(* CODESYS project mpm_jsonparser.library
   Author: Cory Tollefsrud
   Placeholder: MPM_JsonParser
   Title: MPM_JsonParser
   Version: 0.2.3.1
   Company: MatixPM

Project tree, tasks and I/O mapping:
  libraries: Base Interfaces, * (System); Tc2_System, * (Beckhoff Automation GmbH); Tc3_JsonXml, * (Beckhoff Automation GmbH)
  FUN/
    function F_Map_ST_AnyType_User [ST]
  Legecy/
    function block FB_JsonSchemaEx_OLD [ST]: M_CreateSchemaJson, M_PraseSchemaJson, M_PraseJsonSchema, M_SetJsonSchema, M_SetMemberValue, M_SetMemberValue_AnyType, M_SetMemberValueEx, M_SetMemberValueEx_AnyType, M_GetJsonMemberValue, M_GetJsonMemberValue_AnyType, M_SetJsonMember, M_SetJsonMemberValue, M_SetJsonMemberValue_AnyType, M_SetJsonMemberValueEx, M_SetJsonMemberValueEx_AnyType, M_SetJsonMemberValueNonDefault, M_SetJsonSchemaValue
  data type DUT_JsonMemberValue
  data type DUT_JsonSchema
  data type DUT_Pointers
  data type E_TypeClassEx
  function block FB_JsonEx [ST]: M_SetMemberValue, M_SetMemberValueEx, M_GetJsonMemberValue, M_SetJsonMember, M_SetJsonMemberValue, M_SetJsonMemberValueEx, M_SetJsonMemberValueNonDefault
  function block FB_JsonSchemaEx [ST]: M_CreateSchemaJson, M_PraseSchemaJson, M_RegisterSchemaObject
  function block FB_JsonSchemaExBase [ST]: M_AssignSchemaMember, M_AssignSchemaMemberEx, M_GetJsonSchemaValue, M_PraseJsonSchema, M_Read, M_SetJsonSchema, M_SetJsonSchemaValue, M_SetMemberSchemaValue, M_Write
  function block FB_JsonSchemaObject [ST]: M_AssignSchemaMember, M_AssignSchemaMemberEx, M_CreateSchemaJson, M_GetWriteStatus, M_PraseSchemaJson, M_Read, M_SetJsonRef, M_SetJsonSchemaValue, M_TriggerWrite, M_Write, P_sJsonRoot
  data type ST_AnyType_User
  data type ST_SchemaMember
*)

// DUT_JsonMemberValue
TYPE DUT_JsonMemberValue :
STRUCT
	member				: STRING(255);
	value				: STRING(10000);
END_STRUCT
END_TYPE

// DUT_JsonSchema
TYPE DUT_JsonSchema :
STRUCT
	jsonValueRoot			: REFERENCE TO sJsonValue;
	jsonValue				: sJsonValue;
	member					: STRING(255);
	typeClass				: E_TypeClassEx;
END_STRUCT
END_TYPE

// DUT_Pointers
//{attribute 'no_copy'} // used so that on that on a online change the pointers will update there address.

//This is only to copy values in and out of DOM memory
TYPE DUT_Pointers :
STRUCT
	_byteArray			: ARRAY [0..7] OF BYTE;
	pString				: POINTER TO STRING(1000); //String
	pJson				: POINTER TO STRING(10000);	//Big string
	pSint				: POINTER TO SINT;
	pInt				: POINTER TO INT;
	pUInt				: POINTER TO UINT;
	pDint				: POINTER TO DINT;
	pUDint				: POINTER TO UDINT;	
	pLint				: POINTER TO LINT;
	pUlint				: POINTER TO ULINT;	
	pBOOL				: POINTER TO BOOL;
	pLREAL				: POINTER TO LREAL;
	pREAL				: POINTER TO REAL;
	pFileTime			: POINTER TO FILETIME;
END_STRUCT
END_TYPE

// E_TypeClassEx
{attribute 'qualified_only'}

TYPE E_TypeClassEx :
(
	Type_ANY := TypeClass.TYPE_ANY,
	TYPE_ANYBIT := TypeClass.TYPE_ANYBIT,
	TYPE_ANYDATE := TypeClass.TYPE_ANYDATE,
	TYPE_ANYINT := TypeClass.TYPE_ANYINT,	
	TYPE_ANYNUM := TypeClass.TYPE_ANYNUM,	
	TYPE_ANYREAL := TypeClass.TYPE_ANYREAL,		
	TYPE_ARRAY := TypeClass.TYPE_ARRAY,	
	TYPE_BIT := TypeClass.TYPE_BIT,		
	TYPE_BITCONST := TypeClass.TYPE_BITCONST,		
	TYPE_BOOL := TypeClass.TYPE_BOOL,
	TYPE_BYTE := TypeClass.TYPE_BYTE,	
	TYPE_DATE := TypeClass.TYPE_DATE,
	TYPE_DATEANDTIME := TypeClass.TYPE_DATEANDTIME,			
	TYPE_DINT := TypeClass.TYPE_DINT,		
	TYPE_DWORD := TypeClass.TYPE_DWORD,		
	TYPE_ENUM := TypeClass.TYPE_ENUM,	
	TYPE_INT := TypeClass.TYPE_INT,	
	TYPE_INTERFACE := TypeClass.TYPE_INTERFACE,	
	TYPE_LAZY := TypeClass.TYPE_LAZY,		
	TYPE_LINT := TypeClass.TYPE_LINT,
	TYPE_LREAL := TypeClass.TYPE_LREAL,	
	TYPE_LTIME := TypeClass.TYPE_LTIME,	
	TYPE_LWORD := TypeClass.TYPE_LWORD,
	TYPE_NONE := TypeClass.TYPE_NONE,
	TYPE_PARAMS := TypeClass.TYPE_PARAMS,	
	TYPE_POINTER := TypeClass.TYPE_POINTER,	
	TYPE_REAL := TypeClass.TYPE_REAL, 	
	TYPE_REFERENCE := TypeClass.TYPE_REFERENCE,	
	TYPE_SINT := TypeClass.TYPE_SINT,	
	TYPE_STRING := TypeClass.TYPE_STRING,	
	TYPE_SUBRANGE := TypeClass.TYPE_SUBRANGE,
	TYPE_TIME := TypeClass.TYPE_TIME,			
	TYPE_TIMEOFDAY := TypeClass.TYPE_TIMEOFDAY,					
	TYPE_UDINT := TypeClass.TYPE_UDINT,		
	TYPE_UINT := TypeClass.TYPE_UINT,	
	TYPE_ULINT := TypeClass.TYPE_ULINT,
	TYPE_USERDEF := TypeClass.TYPE_USERDEF,	
	TYPE_USINT := TypeClass.TYPE_USINT,	
	TYPE_WORD := TypeClass.TYPE_WORD,	
	TYPE_WSTRING := TypeClass.TYPE_WSTRING,
	TYPE_JSON := 10000,
	TYPE_JSONARRAY := 10002,	
	TYPE_FILETIME := 10001	
)INT;
END_TYPE

// ST_AnyType_User
{attribute 'enable_dynamic_creation'}
TYPE ST_AnyType_User :
STRUCT
	//name
	name : STRING(80);
	// the type of the actual parameter
	typeclass  : E_TypeClassEx ;
      // the pointer to the actual parameter
  	pvalue     : PVOID;
      // the size of the data, to which the pointer points
 	diSize     : DINT;
END_STRUCT
END_TYPE

// ST_SchemaMember
TYPE ST_SchemaMember :
STRUCT
	jsonRoot			: REFERENCE TO SJsonValue;
	member				: STRING(255);
	pValue				: PVOID;
	cbSizeOf			: UDINT;
	eTypeClass			: E_TypeClassEx;	
END_STRUCT
END_TYPE

// FUN/F_Map_ST_AnyType_User
FUNCTION F_Map_ST_AnyType_User : HRESULT
VAR_INPUT
	name : STRING;
	pVar : ANY;
	pst_AnyType_User : REFERENCE TO ST_AnyType_User;
END_VAR
VAR
END_VAR

pst_AnyType_User.diSize := pVar.diSize;
pst_AnyType_User.pValue := pVar.pValue;
pst_AnyType_User.typeclass := TO_INT(pVar.TypeClass);
pst_AnyType_User.name := name;

END_FUNCTION

// Legecy/FB_JsonSchemaEx_OLD
FUNCTION_BLOCK ABSTRACT FB_JsonSchemaEx_OLD EXTENDS FB_JsonDomParser;
VAR_INPUT
END_VAR
VAR_OUTPUT
END_VAR
VAR
	
END_VAR


(*
var
	P_sJsonid			: MPM_JsonParser.DUT_JsonSchema := (member := '_id', typeClass := E_TypeClassEx.TYPE_STRING,jsonValueRoot := jsonRoot);
	P_sJsonTimeStamp	: MPM_JsonParser.DUT_JsonSchema := (member := 'time_stamp', typeClass := E_TypeClassEx.TYPE_FILETIME,jsonValueRoot := jsonRoot);		
	P_sJsonValues		: MPM_JsonParser.DUT_JsonSchema := (member := 'values', typeClass := E_TypeClassEx.TYPE_JSON,jsonValueRoot := jsonRoot);	
	jsonRoot : SJsonValue;	
end_var
*)

METHOD PUBLIC ABSTRACT M_CreateSchemaJson : BOOL
VAR_IN_OUT
END_VAR
(*
jsonRoot := THIS^.NewDocument();
M_SetJsonSchema(jsonRoot,P_sJsonid);
//M_SetJsonSchema(P_sJsonid.jsonValue,P_sJsonRecipe);
M_SetJsonSchema(jsonRoot,P_sJsonValues);
M_SetJsonSchema(jsonRoot,P_sJsonTimeStamp);

*)
END_METHOD

METHOD PUBLIC ABSTRACT M_PraseSchemaJson : BOOL
VAR_INPUT
END_VAR
(*

jsonRoot := THIS^.GetDocumentRoot();
IF jsonRoot > 0 THEN
	M_PraseJsonSchema(jsonRoot,P_sJsonid);
	//M_SetJsonSchema(P_sJsonid.jsonValue,P_sJsonRecipe);
	M_PraseJsonSchema(jsonRoot,P_sJsonValues);
	M_PraseJsonSchema(jsonRoot,P_sJsonTimeStamp);
END_IF


*)
END_METHOD

METHOD PROTECTED M_PraseJsonSchema : sJsonValue //Takes the json schema and finds it in DOM memory and sets its sJsonValue.
VAR_INPUT
	jsonRoot 				: REFERENCE TO sJsonValue;
END_VAR

VAR_IN_OUT
	jsonSchema				: DUT_JsonSchema;
END_VAR
M_PraseJsonSchema := THIS^.FindMember(jsonRoot,jsonSchema.member); //Looks for member
IF M_PraseJsonSchema > 0 THEN //If memeber is found
	jsonSchema.jsonValue := M_PraseJsonSchema;
	jsonSchema.jsonValueRoot REF= jsonRoot;
END_IF
END_METHOD

METHOD PROTECTED M_SetJsonSchema : sJsonValue //Takes a Json Schema variable and adds it to DOM memory. Writes the sJsonValue to json schema.
VAR_INPUT
	jsonRoot 				: REFERENCE TO sJsonValue;
END_VAR

VAR_IN_OUT
	jsonSchema				: DUT_JsonSchema;
END_VAR
CASE jsonSchema.typeClass OF  
	
	E_TypeClassEx.TYPE_JSONARRAY: //Adds an empty array
		jsonSchema.jsonValueRoot REF= jsonRoot;
		jsonSchema.jsonValue := THIS^.AddJsonMember(jsonRoot,jsonSchema.member,'[]');		
		M_SetJsonSchema := jsonSchema.jsonValue;			
	ELSE //Justs sets null value
		jsonSchema.jsonValueRoot REF= jsonRoot;
		jsonSchema.jsonValue := THIS^.AddNullMember(jsonRoot,jsonSchema.member);
		M_SetJsonSchema := jsonSchema.jsonValue;		
END_CASE
END_METHOD

METHOD PROTECTED M_SetMemberValue : sJsonValue //Used to set a member to any type. Has to be a listed type in the TypeClass 
VAR_INPUT
	jsonRoot 	: sJsonValue;
	value			: ANY;
END_VAR
VAR_IN_OUT CONSTANT
	member			: STRING;	
END_VAR
VAR
	pString			: POINTER TO STRING;
	stPointers		: DUT_Pointers;
END_VAR
IF value.TypeClass = E_TypeClassEx.TYPE_ENUM THEN
	CASE value.diSize OF
		4:
			value.TypeClass := E_TypeClassEx.TYPE_INT;
		8:
			value.TypeClass := E_TypeClassEx.TYPE_UDINT;	
	END_CASE
END_IF

CASE value.TypeClass OF 
	E_TypeClassEx.TYPE_STRING:
		pString := value.pValue;
		M_SetMemberValue := THIS^.AddStringMember(jsonRoot,member,pString^);
	E_TypeClassEx.TYPE_LINT:
		stPointers.pLint := value.pValue;
		M_SetMemberValue := THIS^.AddInt64Member(jsonRoot,member,stPointers.pLint^);
	E_TypeClassEx.TYPE_LTIME:
		stPointers.pLint := value.pValue;		
		M_SetMemberValue := THIS^.AddInt64Member(jsonRoot,member,stPointers.pLint^);		
	E_TypeClassEx.TYPE_ULINT:
		stPointers.pUlint := value.pValue;
		M_SetMemberValue := THIS^.AddInt64Member(jsonRoot,member,stPointers.pUlint^);	
	E_TypeClassEx.TYPE_UDINT:
		stPointers.pUDint := value.pValue;		
		M_SetMemberValue := THIS^.AddIntMember(jsonRoot,member,stPointers.pUDint^);
	E_TypeClassEx.TYPE_USINT, E_TypeClassEx.TYPE_SINT:
		stPointers.pSint := value.pValue;		
		M_SetMemberValue := THIS^.AddIntMember(jsonRoot,member,stPointers.pSint^);		
	E_TypeClassEx.TYPE_INT,E_TypeClassEx.TYPE_UINT:
		stPointers.pUInt := value.pValue;	
		M_SetMemberValue := THIS^.AddIntMember(jsonRoot,member,stPointers.pUInt^);		
	E_TypeClassEx.TYPE_DINT, E_TypeClassEx.TYPE_DWORD:
		stPointers.pDint := value.pValue;		
		M_SetMemberValue := THIS^.AddIntMember(jsonRoot,member,stPointers.pDint^);		
	E_TypeClassEx.TYPE_WORD:
		stPointers.pInt := value.pValue;		
		M_SetMemberValue := THIS^.AddIntMember(jsonRoot,member,stPointers.pInt^);		
	E_TypeClassEx.TYPE_REAL:
		stPointers.pREAL := value.pValue;			
		M_SetMemberValue := THIS^.AddDoubleMember(jsonRoot,member,stPointers.pREAL^);
	E_TypeClassEx.TYPE_LREAL:
		stPointers.pLREAL := value.pValue;			
		M_SetMemberValue := THIS^.AddDoubleMember(jsonRoot,member,stPointers.pLREAL^);		
	E_TypeClassEx.TYPE_BOOL:
		stPointers.pBOOL := value.pValue; 
		M_SetMemberValue := THIS^.AddBoolMember(jsonRoot,member,stPointers.pBOOL^);					
END_CASE
END_METHOD

METHOD PROTECTED M_SetMemberValue_AnyType : sJsonValue //Used to set a member to any type. Has to be a listed type in the TypeClass 
VAR_INPUT
	jsonRoot 	: sJsonValue;
	value			: ST_AnyType_User;
END_VAR
VAR_IN_OUT CONSTANT
	member			: STRING;	
END_VAR
VAR
	pString			: POINTER TO STRING;
	stPointers		: DUT_Pointers;
END_VAR
IF value.TypeClass = E_TypeClassEx.TYPE_ENUM THEN
	CASE value.diSize OF
		4:
			value.TypeClass := E_TypeClassEx.TYPE_INT;
		8:
			value.TypeClass := E_TypeClassEx.TYPE_UDINT;	
	END_CASE
END_IF

CASE value.TypeClass OF 
	E_TypeClassEx.TYPE_STRING:
		pString := value.pValue;
		M_SetMemberValue_AnyType := THIS^.AddStringMember(jsonRoot,member,pString^);
	E_TypeClassEx.TYPE_LINT:
		stPointers.pLint := value.pValue;
		M_SetMemberValue_AnyType := THIS^.AddInt64Member(jsonRoot,member,stPointers.pLint^);
	E_TypeClassEx.TYPE_LTIME:
		stPointers.pLint := value.pValue;		
		M_SetMemberValue_AnyType := THIS^.AddInt64Member(jsonRoot,member,stPointers.pLint^);		
	E_TypeClassEx.TYPE_ULINT:
		stPointers.pUlint := value.pValue;
		M_SetMemberValue_AnyType := THIS^.AddInt64Member(jsonRoot,member,stPointers.pUlint^);	
	E_TypeClassEx.TYPE_UDINT:
		stPointers.pUDint := value.pValue;		
		M_SetMemberValue_AnyType := THIS^.AddIntMember(jsonRoot,member,stPointers.pUDint^);
	E_TypeClassEx.TYPE_USINT, E_TypeClassEx.TYPE_SINT:
		stPointers.pSint := value.pValue;		
		M_SetMemberValue_AnyType := THIS^.AddIntMember(jsonRoot,member,stPointers.pSint^);		
	E_TypeClassEx.TYPE_INT,E_TypeClassEx.TYPE_UINT:
		stPointers.pUInt := value.pValue;	
		M_SetMemberValue_AnyType := THIS^.AddIntMember(jsonRoot,member,stPointers.pUInt^);		
	E_TypeClassEx.TYPE_DINT, E_TypeClassEx.TYPE_DWORD:
		stPointers.pDint := value.pValue;		
		M_SetMemberValue_AnyType := THIS^.AddIntMember(jsonRoot,member,stPointers.pDint^);		
	E_TypeClassEx.TYPE_WORD:
		stPointers.pInt := value.pValue;		
		M_SetMemberValue_AnyType := THIS^.AddIntMember(jsonRoot,member,stPointers.pInt^);		
	E_TypeClassEx.TYPE_REAL:
		stPointers.pREAL := value.pValue;			
		M_SetMemberValue_AnyType := THIS^.AddDoubleMember(jsonRoot,member,stPointers.pREAL^);
	E_TypeClassEx.TYPE_LREAL:
		stPointers.pLREAL := value.pValue;			
		M_SetMemberValue_AnyType := THIS^.AddDoubleMember(jsonRoot,member,stPointers.pLREAL^);		
	E_TypeClassEx.TYPE_BOOL:
		stPointers.pBOOL := value.pValue; 
		M_SetMemberValue_AnyType := THIS^.AddBoolMember(jsonRoot,member,stPointers.pBOOL^);					
END_CASE
END_METHOD

METHOD PROTECTED M_SetMemberValueEx : sJsonValue
VAR_INPUT
	jsonValue 	: sJsonValue;
	value		: ANY;
	valueType	: E_TypeClassEx;
END_VAR
VAR
	stPointers		: DUT_Pointers;	
END_VAR
CASE valueType OF 
	E_TypeClassEx.TYPE_FILETIME:
		IF value.diSize = SIZEOF(FILETIME) THEN
			stPointers.pFileTime := value.pValue;
			M_SetMemberValueEx := THIS^.SetFileTime(jsonValue,stPointers.pFileTime^);			
		END_IF	
		E_TypeClassEx.TYPE_JSON:
			stPointers.pJson := value.pValue;
			M_SetMemberValueEx := THIS^.SetJson(jsonValue,stPointers.pJson^);			
END_CASE
END_METHOD

METHOD PROTECTED M_SetMemberValueEx_AnyType : sJsonValue
VAR_INPUT
	jsonValue 	: sJsonValue;
	value		: ST_AnyType_User;
	valueType	: E_TypeClassEx;
END_VAR
VAR
	stPointers		: DUT_Pointers;	
END_VAR
CASE valueType OF 
	E_TypeClassEx.TYPE_FILETIME:
		IF value.diSize = SIZEOF(FILETIME) THEN
			stPointers.pFileTime := value.pValue;
			M_SetMemberValueEx_AnyType := THIS^.SetFileTime(jsonValue,stPointers.pFileTime^);			
		END_IF	
		E_TypeClassEx.TYPE_JSON:
			stPointers.pJson := value.pValue;
			M_SetMemberValueEx_AnyType := THIS^.SetJson(jsonValue,stPointers.pJson^);			
END_CASE
END_METHOD

METHOD PUBLIC M_GetJsonMemberValue : BOOL
VAR_INPUT
	jsonRoot 	: sJsonValue;
END_VAR

VAR_IN_OUT CONSTANT
	member			: STRING;
END_VAR

VAR_INPUT
	value		: ANY;
END_VAR

VAR
END_VAR

VAR
	jsonValue		: sJsonValue;
	stPointers		: DUT_Pointers;	
END_VAR
jsonValue := THIS^.FindMember(jsonRoot,member);

CASE value.TypeClass OF 
	E_TypeClassEx.TYPE_STRING:
		stPointers.pString := value.pValue;
		stPointers.pString^ := THIS^.GetString(jsonValue);
		M_GetJsonMemberValue := TRUE;		
	E_TypeClassEx.TYPE_LINT:
		stPointers.pLint := value.pValue;
		stPointers.pLint^ := THIS^.GetInt64(jsonValue);
		M_GetJsonMemberValue := TRUE;
	E_TypeClassEx.TYPE_ULINT:
		stPointers.pUlint := value.pValue;
		stPointers.pUlint^ := THIS^.GetInt64(jsonValue);	
		M_GetJsonMemberValue := TRUE;		
	E_TypeClassEx.TYPE_UDINT:
		stPointers.pUDint := value.pValue;		
		stPointers.pUDint^ := THIS^.GetInt(jsonValue);			
		M_GetJsonMemberValue := TRUE;	
	 E_TypeClassEx.TYPE_USINT,  E_TypeClassEx.TYPE_SINT:	
		stPointers.pSint := value.pValue;		
		stPointers.pSint^ := TO_SINT(THIS^.GetInt(jsonValue));			
		M_GetJsonMemberValue := TRUE;		 
	E_TypeClassEx.TYPE_DINT, E_TypeClassEx.TYPE_DWORD:
		stPointers.pDint := value.pValue;		
		stPointers.pDint^ := THIS^.GetInt(jsonValue);
		M_GetJsonMemberValue := TRUE;		
	E_TypeClassEx.TYPE_INT, E_TypeClassEx.TYPE_WORD, E_TypeClassEx.TYPE_UINT:
		stPointers.pint := value.pValue;				
		stPointers.pInt^ := TO_INT(THIS^.GetInt(jsonValue));
		M_GetJsonMemberValue := TRUE;		
	E_TypeClassEx.TYPE_REAL:
		stPointers.pREAL := value.pValue;
		stPointers.pReal^ := THIS^.GetDouble(jsonValue);
		M_GetJsonMemberValue := TRUE;
	E_TypeClassEx.TYPE_LREAL:
		stPointers.pLREAL := value.pValue;
		stPointers.pLReal^ := THIS^.GetDouble(jsonValue);
		M_GetJsonMemberValue := TRUE;	
	E_TypeClassEx.TYPE_BOOL:
		stPointers.pBOOL := value.pValue;
		stPointers.pBOOL^ := THIS^.GetBool(jsonValue);	
		M_GetJsonMemberValue := TRUE;				
END_CASE
END_METHOD

METHOD PUBLIC M_GetJsonMemberValue_AnyType : BOOL
VAR_INPUT
	jsonRoot 	: sJsonValue;
END_VAR

VAR_IN_OUT CONSTANT
	member			: STRING;
END_VAR

VAR_INPUT
	value		: ST_AnyType_User;
END_VAR

VAR
END_VAR

VAR
	jsonValue		: sJsonValue;
	stPointers		: DUT_Pointers;	
END_VAR
jsonValue := THIS^.FindMember(jsonRoot,member);

CASE value.TypeClass OF 
	E_TypeClassEx.TYPE_STRING:
		stPointers.pString := value.pValue;
		stPointers.pString^ := THIS^.GetString(jsonValue);
		M_GetJsonMemberValue_AnyType := TRUE;		
	E_TypeClassEx.TYPE_LINT:
		stPointers.pLint := value.pValue;
		stPointers.pLint^ := THIS^.GetInt64(jsonValue);
		M_GetJsonMemberValue_AnyType := TRUE;
	E_TypeClassEx.TYPE_ULINT:
		stPointers.pUlint := value.pValue;
		stPointers.pUlint^ := THIS^.GetInt64(jsonValue);	
		M_GetJsonMemberValue_AnyType := TRUE;		
	E_TypeClassEx.TYPE_UDINT:
		stPointers.pUDint := value.pValue;		
		stPointers.pUDint^ := THIS^.GetInt(jsonValue);			
		M_GetJsonMemberValue_AnyType := TRUE;	
	 E_TypeClassEx.TYPE_USINT,  E_TypeClassEx.TYPE_SINT:	
		stPointers.pSint := value.pValue;		
		stPointers.pSint^ := TO_SINT(THIS^.GetInt(jsonValue));			
		M_GetJsonMemberValue_AnyType := TRUE;		 
	E_TypeClassEx.TYPE_DINT, E_TypeClassEx.TYPE_DWORD:
		stPointers.pDint := value.pValue;		
		stPointers.pDint^ := THIS^.GetInt(jsonValue);
		M_GetJsonMemberValue_AnyType := TRUE;		
	E_TypeClassEx.TYPE_INT, E_TypeClassEx.TYPE_WORD, E_TypeClassEx.TYPE_UINT:
		stPointers.pint := value.pValue;				
		stPointers.pInt^ := TO_INT(THIS^.GetInt(jsonValue));
		M_GetJsonMemberValue_AnyType := TRUE;		
	E_TypeClassEx.TYPE_REAL:
		stPointers.pREAL := value.pValue;
		stPointers.pReal^ := THIS^.GetDouble(jsonValue);
		M_GetJsonMemberValue_AnyType := TRUE;
	E_TypeClassEx.TYPE_LREAL:
		stPointers.pLREAL := value.pValue;
		stPointers.pLReal^ := THIS^.GetDouble(jsonValue);
		M_GetJsonMemberValue_AnyType := TRUE;	
	E_TypeClassEx.TYPE_BOOL:
		stPointers.pBOOL := value.pValue;
		stPointers.pBOOL^ := THIS^.GetBool(jsonValue);	
		M_GetJsonMemberValue_AnyType := TRUE;				
END_CASE
END_METHOD

METHOD PUBLIC M_SetJsonMember : sJsonValue
VAR_INPUT
	jsonRoot 				: sJsonValue;
END_VAR

VAR_IN_OUT CONSTANT
	member				: STRING(255);
END_VAR

VAR
	jsonValue			: sJsonValue;
END_VAR
jsonValue := THIS^.FindMember(jsonRoot,member);

IF jsonValue = 0 THEN
	jsonValue := THIS^.AddNullMember(jsonRoot,member);
	M_SetJsonMember := jsonValue;
ELSE
	M_SetJsonMember := jsonValue;	
END_IF
END_METHOD

METHOD PUBLIC M_SetJsonMemberValue : sJsonValue
VAR_INPUT
	jsonRoot 				: sJsonValue;
END_VAR
VAR_IN_OUT CONSTANT
	member			: STRING;
END_VAR
VAR_INPUT
	value			: ANY;
END_VAR
THIS^.RemoveMemberByName(jsonRoot,member,FALSE);
M_SetJsonMemberValue := M_SetMemberValue(jsonRoot,value,member);
END_METHOD

METHOD PUBLIC M_SetJsonMemberValue_AnyType : sJsonValue
VAR_INPUT
	jsonRoot 				: sJsonValue;
END_VAR
VAR_IN_OUT CONSTANT
	member			: STRING;
END_VAR
VAR_INPUT
	value			: ST_AnyType_User;
END_VAR
THIS^.RemoveMemberByName(jsonRoot,member,FALSE);
M_SetJsonMemberValue_AnyType := M_SetMemberValue_AnyType(jsonRoot,value,member);
END_METHOD

METHOD PUBLIC M_SetJsonMemberValueEx : sJsonValue
VAR_INPUT
	jsonRoot 				: sJsonValue;
END_VAR


VAR_IN_OUT CONSTANT
	member			: STRING;
END_VAR

VAR_INPUT
	value			: ANY;
	valueType		: E_TypeClassEx;		
END_VAR


VAR
	jsonValue		: sJsonValue;
END_VAR
THIS^.RemoveMemberByName(jsonRoot,member,FALSE);

IF jsonValue > 0 THEN	
	IF valueType <> value.TypeClass THEN
		M_SetMemberValueEX(jsonValue,value,valueType);
		M_SetJsonMemberValueEx := jsonValue;
	ELSE
		M_SetJsonMemberValueEx := M_SetMemberValue(jsonRoot,value,member);
	END_IF	
END_IF;
END_METHOD

METHOD PUBLIC M_SetJsonMemberValueEx_AnyType : sJsonValue
VAR_INPUT
	jsonRoot 				: sJsonValue;
END_VAR


VAR_IN_OUT CONSTANT
	member			: STRING;
END_VAR

VAR_INPUT
	value			: ST_AnyType_User;
	valueType		: E_TypeClassEx;		
END_VAR


VAR
	jsonValue		: sJsonValue;
END_VAR
THIS^.RemoveMemberByName(jsonRoot,member,FALSE);

IF jsonValue > 0 THEN	
	IF valueType <> value.TypeClass THEN
		M_SetMemberValueEx_AnyType(jsonValue,value,valueType);
		M_SetJsonMemberValueEx_AnyType := jsonValue;
	ELSE
		M_SetJsonMemberValueEx_AnyType := M_SetMemberValue_AnyType(jsonRoot,value,member);
	END_IF	
END_IF;
END_METHOD

METHOD PUBLIC M_SetJsonMemberValueNonDefault : sJsonValue // Used to allow a condtional check before setting a value. Best use is to check to make sure some value is not zero or some defualt value
VAR_INPUT
	jsonRoot 				: sJsonValue;
END_VAR
VAR_IN_OUT CONSTANT
	member			: STRING;
END_VAR
VAR_INPUT
	value			: ANY;
END_VAR
VAR 
	x				: UDINT;
END_VAR
VAR
	pByte			: POINTER TO BYTE;
	
END_VAR
VAR_OUTPUT
	newValue		: BOOL;
END_VAR
pByte := value.pValue;
FOR x := 0 TO value.diSize - 1 BY SIZEOF(BYTE) DO
	pByte := value.pValue + x;
	IF pByte^ > 0 THEN
		M_SetJsonMemberValueNonDefault := THIS^.M_SetJsonMemberValue(jsonRoot,member,value);
		RETURN;
	END_IF
END_FOR
END_METHOD

METHOD PUBLIC M_SetJsonSchemaValue : sJsonValue
VAR_IN_OUT
	jsonSchema				: DUT_JsonSchema;
END_VAR
VAR_INPUT
	value					: ANY;
END_VAR

VAR
	jsonValue				: sJsonValue;
	pFileTime		: POINTER TO FILETIME;	
	pJson			: POINTER TO STRING(10000);	
END_VAR
jsonValue := THIS^.FindMember(jsonSchema.jsonValueRoot,jsonSchema.member);

IF jsonValue > 0 THEN
	IF jsonSchema.typeClass <> value.TypeClass THEN
		M_SetMemberValueEX(jsonValue,value,jsonSchema.typeClass);
		M_SetJsonSchemaValue := jsonValue;
	ELSE
		M_SetMemberValue(jsonValue,value,jsonSchema.member);
		M_SetJsonSchemaValue := jsonValue;	
	END_IF	
END_IF;
END_METHOD

END_FUNCTION_BLOCK

// FB_JsonEx
FUNCTION_BLOCK FB_JsonEx EXTENDS FB_JsonDomParser;
VAR_INPUT
END_VAR
VAR_OUTPUT
END_VAR
VAR
END_VAR

METHOD PROTECTED M_SetMemberValue : sJsonValue //Used to set a member to any type. Has to be a listed type in the TypeClass 
VAR_INPUT
	jsonRoot 	: sJsonValue;
	value			: ANY;
END_VAR
VAR_IN_OUT CONSTANT
	member			: STRING;	
END_VAR
VAR
	pString			: POINTER TO STRING;
	stPointers		: DUT_Pointers;
END_VAR
IF value.TypeClass = E_TypeClassEx.TYPE_ENUM THEN
	CASE value.diSize OF
		4:
			value.TypeClass := E_TypeClassEx.TYPE_INT;
		8:
			value.TypeClass := E_TypeClassEx.TYPE_UDINT;	
	END_CASE
END_IF

CASE value.TypeClass OF 
	E_TypeClassEx.TYPE_STRING:
		pString := value.pValue;
		M_SetMemberValue := THIS^.AddStringMember(jsonRoot,member,pString^);
	E_TypeClassEx.TYPE_LINT:
		stPointers.pLint := value.pValue;
		M_SetMemberValue := THIS^.AddInt64Member(jsonRoot,member,stPointers.pLint^);
	E_TypeClassEx.TYPE_LTIME:
		stPointers.pLint := value.pValue;		
		M_SetMemberValue := THIS^.AddInt64Member(jsonRoot,member,stPointers.pLint^);		
	E_TypeClassEx.TYPE_ULINT:
		stPointers.pUlint := value.pValue;
		M_SetMemberValue := THIS^.AddInt64Member(jsonRoot,member,stPointers.pUlint^);	
	E_TypeClassEx.TYPE_UDINT:
		stPointers.pUDint := value.pValue;		
		M_SetMemberValue := THIS^.AddIntMember(jsonRoot,member,stPointers.pUDint^);	
	E_TypeClassEx.TYPE_UINT:
		stPointers.pUInt := value.pValue;	
		M_SetMemberValue := THIS^.AddIntMember(jsonRoot,member,stPointers.pUInt^);		
	E_TypeClassEx.TYPE_DINT:
		stPointers.pDint := value.pValue;		
		M_SetMemberValue := THIS^.AddIntMember(jsonRoot,member,stPointers.pDint^);		
	E_TypeClassEx.TYPE_INT:
		stPointers.pInt := value.pValue;		
		M_SetMemberValue := THIS^.AddIntMember(jsonRoot,member,stPointers.pInt^);		
	E_TypeClassEx.TYPE_REAL:
		stPointers.pREAL := value.pValue;			
		M_SetMemberValue := THIS^.AddDoubleMember(jsonRoot,member,stPointers.pREAL^);
	E_TypeClassEx.TYPE_LREAL:
		stPointers.pLREAL := value.pValue;			
		M_SetMemberValue := THIS^.AddDoubleMember(jsonRoot,member,stPointers.pLREAL^);		
	E_TypeClassEx.TYPE_BOOL:
		stPointers.pBOOL := value.pValue; 
		M_SetMemberValue := THIS^.AddBoolMember(jsonRoot,member,stPointers.pBOOL^);					
END_CASE
END_METHOD

METHOD PROTECTED M_SetMemberValueEx : sJsonValue
VAR_INPUT
	jsonValue 	: sJsonValue;
	value		: ANY;
	valueType	: E_TypeClassEx;
END_VAR
VAR
	stPointers		: DUT_Pointers;	
END_VAR
CASE valueType OF 
	E_TypeClassEx.TYPE_FILETIME:
		IF value.diSize = SIZEOF(FILETIME) THEN
			stPointers.pFileTime := value.pValue;
			M_SetMemberValueEx := THIS^.SetFileTime(jsonValue,stPointers.pFileTime^);			
		END_IF	
		E_TypeClassEx.TYPE_JSON:
		IF value.diSize = SIZEOF(FILETIME) THEN
			stPointers.pJson := value.pValue;
			M_SetMemberValueEx := THIS^.SetJson(jsonValue,stPointers.pJson^);			
		END_IF		
END_CASE
END_METHOD

METHOD PUBLIC M_GetJsonMemberValue : BOOL
VAR_INPUT
	jsonRoot 	: sJsonValue;
END_VAR

VAR_IN_OUT CONSTANT
	member			: STRING;
END_VAR

VAR_INPUT
	value		: ANY;
END_VAR

VAR
END_VAR

VAR
	jsonValue		: sJsonValue;
	stPointers		: DUT_Pointers;	
END_VAR
jsonValue := THIS^.FindMember(jsonRoot,member);

CASE value.TypeClass OF 
	E_TypeClassEx.TYPE_STRING:
		stPointers.pString := value.pValue;
		stPointers.pString^ := THIS^.GetString(jsonValue);
		M_GetJsonMemberValue := TRUE;		
	E_TypeClassEx.TYPE_LINT:
		stPointers.pLint := value.pValue;
		stPointers.pLint^ := THIS^.GetInt64(jsonValue);
		M_GetJsonMemberValue := TRUE;
	E_TypeClassEx.TYPE_ULINT:
		stPointers.pUlint := value.pValue;
		stPointers.pUlint^ := THIS^.GetInt64(jsonValue);	
		M_GetJsonMemberValue := TRUE;		
	E_TypeClassEx.TYPE_UDINT:
		stPointers.pUDint := value.pValue;		
		stPointers.pUDint^ := THIS^.GetInt(jsonValue);			
		M_GetJsonMemberValue := TRUE;	
	E_TypeClassEx.TYPE_DINT:
		stPointers.pDint := value.pValue;		
		stPointers.pDint^ := THIS^.GetInt(jsonValue);
		M_GetJsonMemberValue := TRUE;		
	E_TypeClassEx.TYPE_INT:
		stPointers.pint := value.pValue;				
		stPointers.pInt^ := TO_INT(THIS^.GetInt(jsonValue));
		M_GetJsonMemberValue := TRUE;		
	E_TypeClassEx.TYPE_REAL:
		stPointers.pREAL := value.pValue;
		stPointers.pReal^ := THIS^.GetDouble(jsonValue);
		M_GetJsonMemberValue := TRUE;
	E_TypeClassEx.TYPE_LREAL:
		stPointers.pLREAL := value.pValue;
		stPointers.pLReal^ := THIS^.GetDouble(jsonValue);
		M_GetJsonMemberValue := TRUE;	
	E_TypeClassEx.TYPE_BOOL:
		stPointers.pBOOL := value.pValue;
		stPointers.pBOOL^ := THIS^.GetBool(jsonValue);	
		M_GetJsonMemberValue := TRUE;				
END_CASE
END_METHOD

METHOD PUBLIC M_SetJsonMember : sJsonValue
VAR_INPUT
	jsonRoot 				: sJsonValue;
END_VAR

VAR_IN_OUT CONSTANT
	member				: STRING(255);
END_VAR

VAR
	jsonValue			: sJsonValue;
END_VAR
jsonValue := THIS^.FindMember(jsonRoot,member);

IF jsonValue = 0 THEN
	jsonValue := THIS^.AddNullMember(jsonRoot,member);
	M_SetJsonMember := jsonValue;
ELSE
	M_SetJsonMember := jsonValue;	
END_IF
END_METHOD

METHOD PUBLIC M_SetJsonMemberValue : sJsonValue
VAR_INPUT
	jsonRoot 				: sJsonValue;
END_VAR
VAR_IN_OUT CONSTANT
	member			: STRING;
END_VAR
VAR_INPUT
	value			: ANY;
END_VAR
THIS^.RemoveMemberByName(jsonRoot,member,FALSE);
M_SetJsonMemberValue := M_SetMemberValue(jsonRoot,value,member);
END_METHOD

METHOD PUBLIC M_SetJsonMemberValueEx : sJsonValue
VAR_INPUT
	jsonRoot 				: sJsonValue;
END_VAR


VAR_IN_OUT CONSTANT
	member			: STRING;
END_VAR

VAR_INPUT
	value			: ANY;
	valueType		: E_TypeClassEx;		
END_VAR


VAR
	jsonValue		: sJsonValue;
END_VAR
THIS^.RemoveMemberByName(jsonRoot,member,FALSE);

IF jsonValue > 0 THEN	
	IF valueType <> value.TypeClass THEN
		M_SetMemberValueEX(jsonValue,value,valueType);
		M_SetJsonMemberValueEx := jsonValue;
	ELSE
		M_SetJsonMemberValueEx := M_SetMemberValue(jsonRoot,value,member);
	END_IF	
END_IF;
END_METHOD

METHOD PUBLIC M_SetJsonMemberValueNonDefault : sJsonValue // Used to allow a condtional check before setting a value. Best use is to check to make sure some value is not zero or some defualt value
VAR_INPUT
	excute					: BOOL;
	jsonRoot 				: sJsonValue;
END_VAR
VAR_IN_OUT CONSTANT
	member			: STRING;
END_VAR
VAR_INPUT
	value			: ANY;
END_VAR
VAR 
	x				: UDINT;
END_VAR
VAR
	zeroValue		: SINT := 0;
END_VAR
VAR_OUTPUT
	newValue		: BOOL;
END_VAR
IF excute = FALSE THEN
	RETURN;
ELSE
	M_SetJsonMemberValueNonDefault := M_SetJsonMemberValue(jsonRoot,member,value);
END_IF
END_METHOD

END_FUNCTION_BLOCK

// FB_JsonSchemaEx
FUNCTION_BLOCK ABSTRACT FB_JsonSchemaEx EXTENDS FB_JsonSchemaExBase;
VAR_INPUT
	readTrig			: BOOL;
	writeTrig			: BOOL; 		
END_VAR
VAR_OUTPUT
END_VAR
VAR
	jsonRoot			: sJsonValue;
END_VAR

METHOD PUBLIC ABSTRACT M_CreateSchemaJson : BOOL
VAR_IN_OUT
END_VAR
END_METHOD

METHOD PUBLIC ABSTRACT M_PraseSchemaJson : BOOL
VAR_INPUT
END_VAR
END_METHOD

METHOD PUBLIC M_RegisterSchemaObject : BOOL
VAR_INPUT
	fbSchema			: REFERENCE TO FB_JsonSchemaObject;
END_VAR
VAR_IN_OUT
	sJsonRoot			: sJsonValue;
END_VAR
fbSchema.M_SetJsonRef(THIS^,sJsonRoot,writeTrig,readTrig);
//fbSchema.P_sJsonRoot REF= sJsonRoot;
END_METHOD

END_FUNCTION_BLOCK

// FB_JsonSchemaExBase
FUNCTION_BLOCK ABSTRACT FB_JsonSchemaExBase EXTENDS FB_JsonEx 
VAR_INPUT
END_VAR
VAR_OUTPUT
END_VAR
VAR

END_VAR

METHOD PUBLIC M_AssignSchemaMember : BOOL
VAR_IN_OUT
	jsonRoot			: SJsonValue;	
	a_stJsonSchema		: ST_SchemaMember;	
END_VAR
VAR_IN_OUT CONSTANT
	member				: STRING(255);
END_VAR
VAR_INPUT
	value				: ANY;
END_VAR
a_stJsonSchema.jsonRoot REF= jsonRoot;
a_stJsonSchema.member := member;
a_stJsonSchema.pValue := value.pValue;
a_stJsonSchema.cbSizeOf := value.diSize;
a_stJsonSchema.eTypeClass := TO_INT(value.TypeClass);
END_METHOD

METHOD PUBLIC M_AssignSchemaMemberEx : BOOL
VAR_IN_OUT
	jsonRoot			: SJsonValue;
	a_stJsonSchema		: ST_SchemaMember;	
END_VAR
VAR_IN_OUT CONSTANT
	member				: STRING(255);
END_VAR
VAR_INPUT
	value				: ANY;
	eTypeClass			: E_TypeClassEx;
END_VAR
a_stJsonSchema.jsonRoot REF= jsonRoot;
a_stJsonSchema.member := member;
a_stJsonSchema.pValue := value.pValue;
a_stJsonSchema.cbSizeOf := value.diSize;
a_stJsonSchema.eTypeClass := eTypeClass;
END_METHOD

METHOD PROTECTED M_GetJsonSchemaValue : BOOL
VAR_IN_OUT
	a_stJsonSchema		: ST_SchemaMember;	
END_VAR
VAR
	stPointers		: DUT_Pointers;	
END_VAR
CASE a_stJsonSchema.eTypeClass OF 
	E_TypeClassEx.TYPE_STRING:
		stPointers.pString := a_stJsonSchema.pValue;
		stPointers.pString^ := THIS^.GetString(a_stJsonSchema.jsonRoot);
		M_GetJsonSchemaValue := TRUE;		
	E_TypeClassEx.TYPE_LINT:
		stPointers.pLint := a_stJsonSchema.pValue;
		stPointers.pLint^ := THIS^.GetInt64(a_stJsonSchema.jsonRoot);
		M_GetJsonSchemaValue := TRUE;
	E_TypeClassEx.TYPE_ULINT:
		stPointers.pUlint := a_stJsonSchema.pValue;
		stPointers.pUlint^ := THIS^.GetInt64(a_stJsonSchema.jsonRoot);	
		M_GetJsonSchemaValue := TRUE;		
	E_TypeClassEx.TYPE_UDINT:
		stPointers.pUDint := a_stJsonSchema.pValue;		
		stPointers.pUDint^ := THIS^.GetInt(a_stJsonSchema.jsonRoot);			
		M_GetJsonSchemaValue := TRUE;	
	E_TypeClassEx.TYPE_DINT:
		stPointers.pDint := a_stJsonSchema.pValue;		
		stPointers.pDint^ := THIS^.GetInt(a_stJsonSchema.jsonRoot);
		M_GetJsonSchemaValue := TRUE;		
	E_TypeClassEx.TYPE_INT:
		stPointers.pint := a_stJsonSchema.pValue;				
		stPointers.pInt^ := TO_INT(THIS^.GetInt(a_stJsonSchema.jsonRoot));
		M_GetJsonSchemaValue := TRUE;		
	E_TypeClassEx.TYPE_REAL:
		stPointers.pREAL := a_stJsonSchema.pValue;
		stPointers.pReal^ := THIS^.GetDouble(a_stJsonSchema.jsonRoot);
		M_GetJsonSchemaValue := TRUE;
	E_TypeClassEx.TYPE_LREAL:
		stPointers.pLREAL := a_stJsonSchema.pValue;
		stPointers.pLReal^ := THIS^.GetDouble(a_stJsonSchema.jsonRoot);
		M_GetJsonSchemaValue := TRUE;	
	E_TypeClassEx.TYPE_BOOL:
		stPointers.pBOOL := a_stJsonSchema.pValue;
		stPointers.pBOOL^ := THIS^.GetBool(a_stJsonSchema.jsonRoot);	
		M_GetJsonSchemaValue := TRUE;				
END_CASE
END_METHOD

METHOD PUBLIC M_PraseJsonSchema : sJsonValue //Takes the json schema and finds it in DOM memory and sets its sJsonValue.
VAR_INPUT
	jsonRoot 				: sJsonValue;
END_VAR

VAR_IN_OUT
	jsonSchema				: DUT_JsonSchema;
END_VAR
M_PraseJsonSchema := THIS^.FindMember(jsonRoot,jsonSchema.member); //Looks for member
IF M_PraseJsonSchema > 0 THEN //If memeber is found
	jsonSchema.jsonValue := M_PraseJsonSchema;
	jsonSchema.jsonValueRoot := jsonRoot;
END_IF
END_METHOD

METHOD PUBLIC FINAL M_Read : BOOL
VAR_IN_OUT
	a_stJsonSchema		: ARRAY [*] OF ST_SchemaMember;	
END_VAR
VAR
	x							: DINT;
END_VAR
FOR x := LOWER_BOUND(a_stJsonSchema,1) TO UPPER_BOUND(a_stJsonSchema,1) BY 1 DO
	IF __ISVALIDREF(a_stJsonSchema[x].jsonRoot) = FALSE  OR a_stJsonSchema[x].pValue = 0 THEN
		EXIT;
	END_IF	
	M_Read := M_GetJsonSchemaValue(a_stJsonSchema[x]);
END_FOR
END_METHOD

METHOD PUBLIC M_SetJsonSchema : sJsonValue //Takes a Json Schema variable and adds it to DOM memory. Writes the sJsonValue to json schema.
VAR_INPUT
	jsonRoot 				: REFERENCE TO sJsonValue;
END_VAR

VAR_IN_OUT
	jsonSchema				: DUT_JsonSchema;
END_VAR
CASE jsonSchema.typeClass OF  
	
	E_TypeClassEx.TYPE_JSONARRAY: //Adds an empty array
		jsonSchema.jsonValueRoot REF= jsonRoot;
		jsonSchema.jsonValue := THIS^.AddJsonMember(jsonRoot,jsonSchema.member,'[]');		
		M_SetJsonSchema := jsonSchema.jsonValue;			
	ELSE //Justs sets null value
		jsonSchema.jsonValueRoot REF= jsonRoot;
		jsonSchema.jsonValue := THIS^.AddNullMember(jsonRoot,jsonSchema.member);
		M_SetJsonSchema := jsonSchema.jsonValue;		
END_CASE
END_METHOD

METHOD PUBLIC M_SetJsonSchemaValue : sJsonValue
VAR_IN_OUT
	jsonSchema				: DUT_JsonSchema;
END_VAR
VAR_INPUT
	value					: ANY;
END_VAR

VAR
	jsonValue				: sJsonValue;
	pFileTime		: POINTER TO FILETIME;	
	pJson			: POINTER TO STRING(10000);	
END_VAR
jsonValue := THIS^.FindMember(jsonSchema.jsonValueRoot,jsonSchema.member);

IF jsonValue > 0 THEN
	IF jsonSchema.typeClass <> value.TypeClass THEN
		M_SetMemberValueEX(jsonValue,value,jsonSchema.typeClass);
		M_SetJsonSchemaValue := jsonValue;
	ELSE
		M_SetMemberValue(jsonValue,value,jsonSchema.member);
		M_SetJsonSchemaValue := jsonValue;	
	END_IF	
END_IF;
END_METHOD

METHOD PROTECTED M_SetMemberSchemaValue : sJsonValue //Used to set a member to any type. Has to be a listed type in the TypeClass 
VAR_IN_OUT
	a_stJsonSchema		: ST_SchemaMember;	
END_VAR
VAR
	stPointers		: DUT_Pointers;			
END_VAR


CASE a_stJsonSchema.eTypeClass OF 
	E_TypeClassEx.TYPE_STRING:
		stPointers.pString := a_stJsonSchema.pValue;
		M_SetMemberSchemaValue := THIS^.AddStringMember(a_stJsonSchema.jsonRoot,a_stJsonSchema.member,stPointers.pString^);
	E_TypeClassEx.TYPE_LINT:
		stPointers.pLint := a_stJsonSchema.pValue;
		M_SetMemberSchemaValue := THIS^.AddInt64Member(a_stJsonSchema.jsonRoot,a_stJsonSchema.member,stPointers.pLint^);
	E_TypeClassEx.TYPE_LTIME:	
		stPointers.pLint := a_stJsonSchema.pValue;	
		M_SetMemberSchemaValue := THIS^.AddInt64Member(a_stJsonSchema.jsonRoot,a_stJsonSchema.member,stPointers.pLint^);		
	E_TypeClassEx.TYPE_ULINT:
		stPointers.pULint := a_stJsonSchema.pValue;		
		M_SetMemberSchemaValue := THIS^.AddInt64Member(a_stJsonSchema.jsonRoot,a_stJsonSchema.member,stPointers.pULint^);	
	E_TypeClassEx.TYPE_UDINT:		
		stPointers.pUDint := a_stJsonSchema.pValue;		
		M_SetMemberSchemaValue := THIS^.AddIntMember(a_stJsonSchema.jsonRoot,a_stJsonSchema.member,stPointers.pUDint^);	
	E_TypeClassEx.TYPE_UINT:
		stPointers.pUint := a_stJsonSchema.pValue;			
		M_SetMemberSchemaValue := THIS^.AddIntMember(a_stJsonSchema.jsonRoot,a_stJsonSchema.member,stPointers.pUint^);		
	E_TypeClassEx.TYPE_DINT:
		stPointers.pDint := a_stJsonSchema.pValue;		
		M_SetMemberSchemaValue := THIS^.AddIntMember(a_stJsonSchema.jsonRoot,a_stJsonSchema.member,stPointers.pDint^);		
	E_TypeClassEx.TYPE_INT:		
		stPointers.pInt := a_stJsonSchema.pValue;		
		M_SetMemberSchemaValue := THIS^.AddIntMember(a_stJsonSchema.jsonRoot,a_stJsonSchema.member,stPointers.pInt^);		
	E_TypeClassEx.TYPE_REAL:		
		stPointers.pREAL := a_stJsonSchema.pValue;
		M_SetMemberSchemaValue := THIS^.AddDoubleMember(a_stJsonSchema.jsonRoot,a_stJsonSchema.member,stPointers.pREAL^);
	E_TypeClassEx.TYPE_LREAL:	
		stPointers.pLREAL := a_stJsonSchema.pValue;		
		M_SetMemberSchemaValue := THIS^.AddDoubleMember(a_stJsonSchema.jsonRoot,a_stJsonSchema.member,stPointers.pLREAL^);		
	E_TypeClassEx.TYPE_BOOL:
		stPointers.pBOOL := a_stJsonSchema.pValue;	
		M_SetMemberSchemaValue := THIS^.AddBoolMember(a_stJsonSchema.jsonRoot,a_stJsonSchema.member,stPointers.pBOOL^);					
END_CASE
END_METHOD

METHOD PUBLIC FINAL M_Write : SJsonValue
VAR_IN_OUT
	a_stJsonSchema		: ARRAY [*] OF ST_SchemaMember;	
END_VAR
VAR
	x							: DINT;
	isTrue						: BOOL;
END_VAR
FOR x := LOWER_BOUND(a_stJsonSchema,1) TO UPPER_BOUND(a_stJsonSchema,1) BY 1 DO
	isTrue :=  __ISVALIDREF(a_stJsonSchema[x].jsonRoot);
	isTRue := a_stJsonSchema[x].pValue = 0;
	IF __ISVALIDREF(a_stJsonSchema[x].jsonRoot) = FALSE  OR a_stJsonSchema[x].pValue = 0 THEN
		EXIT;
	END_IF
	M_Write := M_SetMemberSchemaValue(a_stJsonSchema[x]);
END_FOR
END_METHOD

END_FUNCTION_BLOCK

// FB_JsonSchemaObject
FUNCTION_BLOCK FB_JsonSchemaObject
VAR_INPUT
END_VAR
VAR_OUTPUT
END_VAR
VAR
	jsonRef				: REFERENCE TO FB_JsonSchemaEx;	
	jsonRoot			: REFERENCE TO SJsonValue;
	read				: BOOL;
	write				: BOOL;
	readTrigREF			: REFERENCE TO BOOL;
	writeTrigREF		: REFERENCE TO BOOL; 		
END_VAR

METHOD PUBLIC M_AssignSchemaMember : BOOL
VAR_IN_OUT
	jsonRoot			: SJsonValue;	
	a_stJsonSchema		: ST_SchemaMember;	
END_VAR
VAR_IN_OUT CONSTANT
	member				: STRING(255);
END_VAR
VAR_INPUT
	value				: ANY;
END_VAR
IF __ISVALIDREF(jsonRef) THEN
	M_AssignSchemaMember := jsonRef.M_AssignSchemaMember(jsonRoot,a_stJsonSchema,member,value);
END_IF
END_METHOD

METHOD PUBLIC M_AssignSchemaMemberEx : BOOL
VAR_IN_OUT
	jsonRoot			: SJsonValue;
	a_stJsonSchema		: ST_SchemaMember;	
END_VAR
VAR_IN_OUT CONSTANT
	member				: STRING(255);
END_VAR
VAR_INPUT
	value				: ANY;
	eTypeClass			: E_TypeClassEx;
END_VAR
IF __ISVALIDREF(jsonRef) THEN
	M_AssignSchemaMemberEx := jsonRef.M_AssignSchemaMemberEx(jsonRoot,a_stJsonSchema,member,value,eTypeClass);
END_IF
END_METHOD

METHOD PUBLIC M_CreateSchemaJson : BOOL
VAR_IN_OUT
	a_stJsonSchema			: ARRAY [*] OF DUT_JsonSchema;
END_VAR

VAR
	x				: DINT;
END_VAR
IF __ISVALIDREF(jsonRef) THEN 
	FOR x := LOWER_BOUND(a_stJsonSchema,1) TO UPPER_BOUND(a_stJsonSchema,1) BY 1 DO
		jsonRef.M_SetJsonSchema(a_stJsonSchema[x].jsonValueRoot,a_stJsonSchema[x]);
	END_FOR
END_IF
END_METHOD

METHOD PUBLIC M_GetWriteStatus : BOOL
VAR_INPUT
END_VAR
IF __ISVALIDREF(writeTrigREF) = TRUE THEN
	M_GetWriteStatus := writeTrigREF;
END_IF
END_METHOD

METHOD PUBLIC M_PraseSchemaJson : BOOL
VAR_IN_OUT
	a_stJsonSchema			: ARRAY [*] OF DUT_JsonSchema;
END_VAR

VAR
	x				: DINT;
END_VAR
IF __ISVALIDREF(jsonRef) THEN 
	FOR x := LOWER_BOUND(a_stJsonSchema,1) TO UPPER_BOUND(a_stJsonSchema,1) BY 1 DO
		jsonRef.M_SetJsonSchema(a_stJsonSchema[x].jsonValueRoot,a_stJsonSchema[x]);
	END_FOR
END_IF
END_METHOD

METHOD PUBLIC FINAL M_Read : BOOL
VAR_IN_OUT
	a_stJsonSchema		: ARRAY [*] OF ST_SchemaMember;	
END_VAR
IF __ISVALIDREF(jsonRef) = FALSE THEN
	RETURN;
END_IF

IF readTrigREF = TRUE AND read = FALSE THEN
	M_Read := jsonRef.M_Read(a_stJsonSchema);
	read := TRUE;
END_IF	

IF readTrigREF = TRUE AND read = FALSE THEN
	M_Read := jsonRef.M_Read(a_stJsonSchema);
	read := TRUE;
END_IF
END_METHOD

METHOD INTERNAL M_SetJsonRef : BOOL
VAR_INPUT
	jsonSchema		: REFERENCE TO FB_JsonSchemaEx;
	jsonRoot		: REFERENCE TO sJsonValue;
	writeRef		: REFERENCE TO BOOL;
	readRef			: REFERENCE TO BOOL;
END_VAR
jsonRef REF= jsonSchema;
THIS^.jsonRoot REF= jsonRoot;
THIS^.readTrigREF REF= readRef;
THIS^.writeTrigREF REF= writeRef;
END_METHOD

METHOD PUBLIC M_SetJsonSchemaValue : sJsonValue
VAR_IN_OUT
	jsonSchema				: DUT_JsonSchema;
END_VAR
VAR_INPUT
	value					: ANY;
END_VAR
IF __ISVALIDREF(jsonRef) THEN
	M_SetJsonSchemaValue := jsonRef.M_SetJsonSchemaValue(jsonSchema,value);
END_IF
END_METHOD

METHOD PUBLIC M_TriggerWrite : BOOL
VAR_INPUT
END_VAR
IF __ISVALIDREF(writeTrigREF) = TRUE THEN
	writeTrigREF := TRUE;
END_IF
END_METHOD

METHOD PUBLIC FINAL M_Write : SJsonValue
VAR_IN_OUT
	a_stJsonSchema		: ARRAY [*] OF ST_SchemaMember;	
END_VAR
IF __ISVALIDREF(jsonRef) = FALSE THEN
	RETURN;
END_IF

IF writeTrigREF = TRUE AND write = FALSE THEN
	M_Write := jsonRef.M_Write(a_stJsonSchema);
	write	:= TRUE;
END_IF	

IF writeTrigREF = FALSE THEN
	write	:= FALSE;
END_IF
END_METHOD

PROPERTY PUBLIC P_sJsonRoot : REFERENCE TO  sJsonValue
GET
P_sJsonRoot REF= jsonRoot;
END_GET
END_PROPERTY

END_FUNCTION_BLOCK
